// TIA Portal V19 export
DATA_BLOCK "instSimulation"   // DB138
// stored: InstanceOfName Unit2.Em6.Simulation, InstanceOfType FB, Namespace Unit2.Em6
"Unit2.Em6.Simulation"
   // VAR
   //    scenario { ExternalWritable := 'False'} : Int;
   //    singleStep { ExternalWritable := 'False'} : Bool;
   //    nextStep { ExternalWritable := 'False'} : Bool;
   //    start { ExternalWritable := 'False'} : Bool;
   //    stop { ExternalWritable := 'False'} : Bool;
   //    stepCounter { ExternalWritable := 'False'} : Int;
   //    nextStepCounter { ExternalWritable := 'False'} : Int;
   //    timer1 { ExternalWritable := 'False'} : TON_TIME;
   //    instR_TRIG { ExternalWritable := 'False'; S7_SetPoint := 'True'} : R_TRIG;
   //    timer1_PT { ExternalWritable := 'False'; S7_SetPoint := 'True'} : Time;
   //    lstPosAbsoluteBusy { ExternalWritable := 'False'} : Bool;
   //    I { ExternalAccessible := 'False'; ExternalVisible := 'False'; ExternalWritable := 'False'} : DInt;
   //    timer1_in { ExternalAccessible := 'False'; ExternalVisible := 'False'; ExternalWritable := 'False'} : Bool;
   //    lstStart { ExternalWritable := 'False'} : Bool;
   // END_VAR
BEGIN
END_DATA_BLOCK
